FUNCTION_BLOCK FB_TelescopeInitializingState EXTENDS FB_TelescopeState
VAR_INPUT
END_VAR
VAR_OUTPUT
END_VAR
VAR
END_VAR

// 
// state
//

// run until initialized
IF NOT fbMachine.pControl^._Initialize() THEN
	fbMachine.State := E_TelescopeState.idle;
END_IF

END_FUNCTION_BLOCK

(* stored: Version 1.1.0.1, ProductVersion 3.1.4024.15
   POU FB_TelescopeInitializingState: Id {10605cd4-f7cc-4286-ab4b-dec57477668d}, SpecialFunc None *)
